FUNCTION_BLOCK ASRT_AX_CLIENT_0_SUBSCRIBE_1 (* Trigger 3 independent remote OPC-UA method calls via CLIENT_0 (Set/Reset/Toggle) and read the resulting state back via SUBSCRIBE_1, driven by an ASRT_AX bidirectional adapter Socket *)
  (* Standard: 61499-2; Description: Copyright (c) 2026 HR Agrartechnik GmbH This program and the accompanying materials are made available under the terms of the Eclipse Public License 2.0 which is available at https://www.eclipse.org/legal/epl-2.0/ SPDX-License-Identifier: EPL-2.0 *)
  (* Version 1.0, 2026-09-03, Franz Höpfinger, HR Agrartechnik GmbH, initial API and implementation and/or initial documentation *)
  PACKAGE adapter::net;
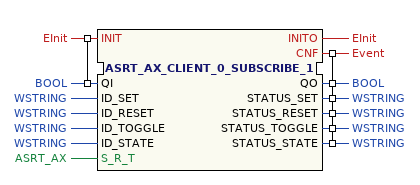
  EVENT_INPUT
    INIT : EInit WITH QI; (* Initialization *)
  END_EVENT
  EVENT_OUTPUT
    INITO : EInit; (* Initialization Confirm *)
    CNF WITH QO, STATUS_SET, STATUS_RESET, STATUS_TOGGLE, STATUS_STATE; (* QO/STATUS updated *)
  END_EVENT
  VAR_INPUT
    QI : BOOL;
    ID_SET : WSTRING; (* Remote-Methodenadresse fuer den Set-Aufruf *)
    ID_RESET : WSTRING; (* Remote-Methodenadresse fuer den Reset-Aufruf *)
    ID_TOGGLE : WSTRING; (* Remote-Methodenadresse fuer den Toggle-Aufruf *)
    ID_STATE : WSTRING; (* Lokal ueberwachter Zustandsknoten (ACTION=READ) *)
  END_VAR
  VAR_OUTPUT
    QO : BOOL; (* TRUE nur wenn SET_CLIENT, RESET_CLIENT, TOGGLE_CLIENT und STATE_SUBSCRIBE aktuell alle QO=TRUE melden *)
    STATUS_SET : WSTRING; (* STATUS von SET_CLIENT *)
    STATUS_RESET : WSTRING; (* STATUS von RESET_CLIENT *)
    STATUS_TOGGLE : WSTRING; (* STATUS von TOGGLE_CLIENT *)
    STATUS_STATE : WSTRING; (* STATUS von STATE_SUBSCRIBE *)
  END_VAR
  SOCKETS
    S_R_T : adapter::types::bidirectional::ASRT_AX; (* Set/Reset/Toggle (out), Zustand (in) *)
  END_SOCKETS
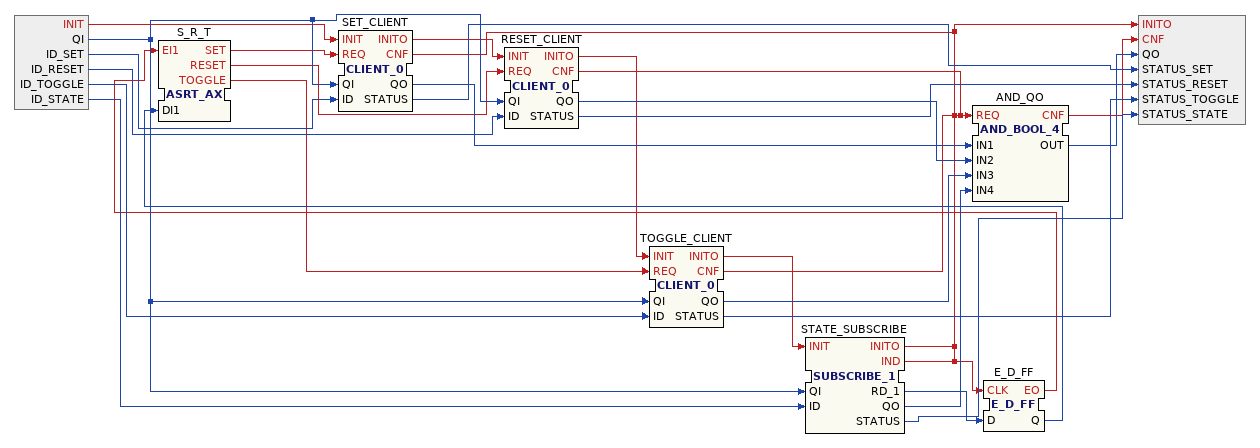
  FBS
    SET_CLIENT : iec61499::net::CLIENT_0;
    RESET_CLIENT : iec61499::net::CLIENT_0;
    TOGGLE_CLIENT : iec61499::net::CLIENT_0;
    STATE_SUBSCRIBE : iec61499::net::SUBSCRIBE_1;
    E_D_FF : iec61499::events::E_D_FF;
    AND_QO : iec61131::booleanOperators::AND_BOOL_4;
  END_FBS
  EVENT_CONNECTIONS
    INIT TO SET_CLIENT.INIT;
    SET_CLIENT.INITO TO RESET_CLIENT.INIT;
    RESET_CLIENT.INITO TO TOGGLE_CLIENT.INIT;
    TOGGLE_CLIENT.INITO TO STATE_SUBSCRIBE.INIT;
    STATE_SUBSCRIBE.INITO TO INITO;
    STATE_SUBSCRIBE.INITO TO AND_QO.REQ;
    S_R_T.SET TO SET_CLIENT.REQ;
    S_R_T.RESET TO RESET_CLIENT.REQ;
    S_R_T.TOGGLE TO TOGGLE_CLIENT.REQ;
    STATE_SUBSCRIBE.IND TO E_D_FF.CLK;
    E_D_FF.EO TO S_R_T.EI1;
    SET_CLIENT.CNF TO AND_QO.REQ;
    RESET_CLIENT.CNF TO AND_QO.REQ;
    TOGGLE_CLIENT.CNF TO AND_QO.REQ;
    STATE_SUBSCRIBE.IND TO AND_QO.REQ;
    AND_QO.CNF TO CNF;
  END_CONNECTIONS
  DATA_CONNECTIONS
    QI TO SET_CLIENT.QI;
    QI TO RESET_CLIENT.QI;
    QI TO TOGGLE_CLIENT.QI;
    QI TO STATE_SUBSCRIBE.QI;
    ID_SET TO SET_CLIENT.ID;
    ID_RESET TO RESET_CLIENT.ID;
    ID_TOGGLE TO TOGGLE_CLIENT.ID;
    ID_STATE TO STATE_SUBSCRIBE.ID;
    STATE_SUBSCRIBE.RD_1 TO E_D_FF.D;
    E_D_FF.Q TO S_R_T.DI1;
    SET_CLIENT.QO TO AND_QO.IN1;
    RESET_CLIENT.QO TO AND_QO.IN2;
    TOGGLE_CLIENT.QO TO AND_QO.IN3;
    STATE_SUBSCRIBE.QO TO AND_QO.IN4;
    AND_QO.OUT TO QO;
    SET_CLIENT.STATUS TO STATUS_SET;
    RESET_CLIENT.STATUS TO STATUS_RESET;
    TOGGLE_CLIENT.STATUS TO STATUS_TOGGLE;
    STATE_SUBSCRIBE.STATUS TO STATUS_STATE;
  END_CONNECTIONS
END_FUNCTION_BLOCK
